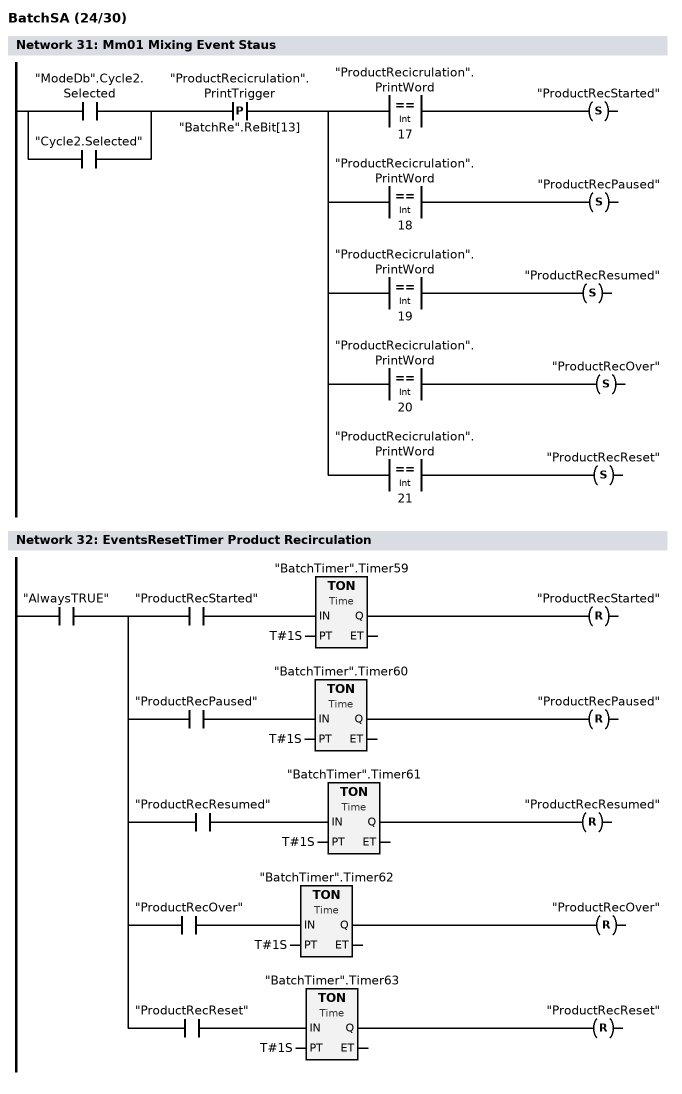
   RUNG wire#powerrail
      Contact( "ModeDb".Cycle2.Selected )
      wire#w1
      P_Contact(operand := "ProductRecicrulation".PrintTrigger, bit := "BatchRe".ReBit[13])
      wire#w2
      { S7_Templates := "SrcType := Int" } EQ_Contact(in1 := "ProductRecicrulation".PrintWord, in2 := 17)
      S_Coil( "ProductRecStarted" )
   END_RUNG
   RUNG wire#powerrail
      Contact( "Cycle2.Selected" )
   END_RUNG wire#w1
   RUNG wire#w2
      { S7_Templates := "SrcType := Int" } EQ_Contact(in1 := "ProductRecicrulation".PrintWord, in2 := 18)
      S_Coil( "ProductRecPaused" )
   END_RUNG
   RUNG wire#w2
      { S7_Templates := "SrcType := Int" } EQ_Contact(in1 := "ProductRecicrulation".PrintWord, in2 := 19)
      S_Coil( "ProductRecResumed" )
   END_RUNG
   RUNG wire#w2
      { S7_Templates := "SrcType := Int" } EQ_Contact(in1 := "ProductRecicrulation".PrintWord, in2 := 20)
      S_Coil( "ProductRecOver" )
   END_RUNG
   RUNG wire#w2
      { S7_Templates := "SrcType := Int" } EQ_Contact(in1 := "ProductRecicrulation".PrintWord, in2 := 21)
      S_Coil( "ProductRecReset" )
   END_RUNG
   // the same network as SCL:
   #_w1 := ("ModeDb".Cycle2.Selected OR "Cycle2.Selected") AND "ProductRecicrulation".PrintTrigger AND NOT "BatchRe".ReBit[13];   // rising edge of "ProductRecicrulation".PrintTrigger
   "BatchRe".ReBit[13] := "ProductRecicrulation".PrintTrigger;
   IF #_w1 AND ("ProductRecicrulation".PrintWord = 17) THEN "ProductRecStarted" := TRUE; END_IF;
   IF #_w1 AND ("ProductRecicrulation".PrintWord = 18) THEN "ProductRecPaused" := TRUE; END_IF;
   IF #_w1 AND ("ProductRecicrulation".PrintWord = 19) THEN "ProductRecResumed" := TRUE; END_IF;
   IF #_w1 AND ("ProductRecicrulation".PrintWord = 20) THEN "ProductRecOver" := TRUE; END_IF;
   IF #_w1 AND ("ProductRecicrulation".PrintWord = 21) THEN "ProductRecReset" := TRUE; END_IF;
END_REGION

REGION Network 32: EventsResetTimer Product Recirculation
   RUNG wire#powerrail
      Contact( "AlwaysTRUE" )
      wire#w1
      Contact( "ProductRecStarted" )
      { S7_Templates := "time_type := Time" } "BatchTimer".Timer59.TON(pt := T#1S, et =>)
      R_Coil( "ProductRecStarted" )
   END_RUNG
   RUNG wire#w1
      Contact( "ProductRecPaused" )
      { S7_Templates := "time_type := Time" } "BatchTimer".Timer60.TON(pt := T#1S, et =>)
      R_Coil( "ProductRecPaused" )
   END_RUNG
   RUNG wire#w1
      Contact( "ProductRecResumed" )
      { S7_Templates := "time_type := Time" } "BatchTimer".Timer61.TON(pt := T#1S, et =>)
      R_Coil( "ProductRecResumed" )
   END_RUNG
   RUNG wire#w1
      Contact( "ProductRecOver" )
      { S7_Templates := "time_type := Time" } "BatchTimer".Timer62.TON(pt := T#1S, et =>)
      R_Coil( "ProductRecOver" )
   END_RUNG
   RUNG wire#w1
      Contact( "ProductRecReset" )
      { S7_Templates := "time_type := Time" } "BatchTimer".Timer63.TON(pt := T#1S, et =>)
      R_Coil( "ProductRecReset" )
   END_RUNG
   // the same network as SCL:
   "BatchTimer".Timer59.TON(IN := "AlwaysTRUE" AND "ProductRecStarted", PT := T#1S);
   IF "BatchTimer".Timer59.Q THEN "ProductRecStarted" := FALSE; END_IF;
   "BatchTimer".Timer60.TON(IN := "AlwaysTRUE" AND "ProductRecPaused", PT := T#1S);
   IF "BatchTimer".Timer60.Q THEN "ProductRecPaused" := FALSE; END_IF;
   "BatchTimer".Timer61.TON(IN := "AlwaysTRUE" AND "ProductRecResumed", PT := T#1S);
   IF "BatchTimer".Timer61.Q THEN "ProductRecResumed" := FALSE; END_IF;
   "BatchTimer".Timer62.TON(IN := "AlwaysTRUE" AND "ProductRecOver", PT := T#1S);
   IF "BatchTimer".Timer62.Q THEN "ProductRecOver" := FALSE; END_IF;
   "BatchTimer".Timer63.TON(IN := "AlwaysTRUE" AND "ProductRecReset", PT := T#1S);
   IF "BatchTimer".Timer63.Q THEN "ProductRecReset" := FALSE; END_IF;
END_REGION

REGION Network 33: EventsResetTimer FIill PWI
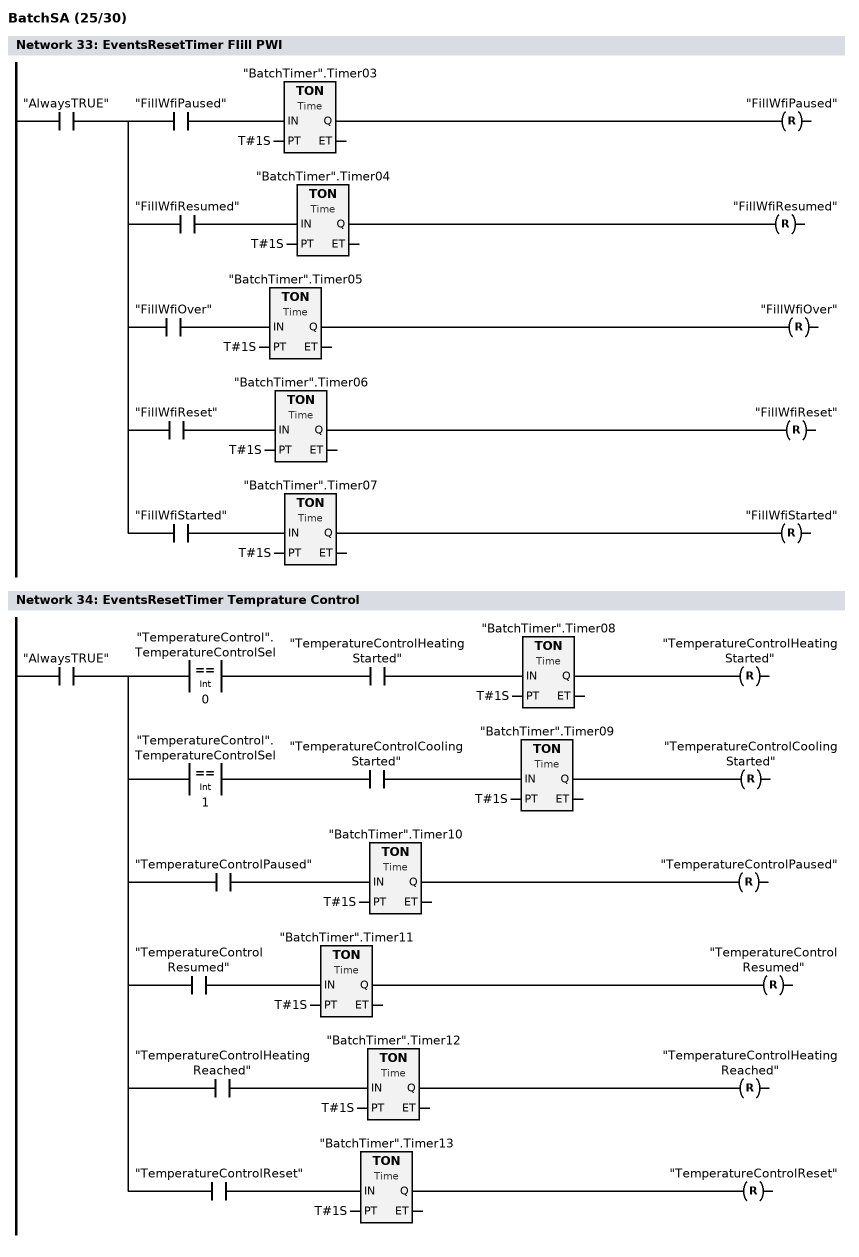
   RUNG wire#powerrail
      Contact( "AlwaysTRUE" )
      wire#w1
      Contact( "FillWfiPaused" )
      { S7_Templates := "time_type := Time" } "BatchTimer".Timer03.TON(pt := T#1S, et =>)
      R_Coil( "FillWfiPaused" )
   END_RUNG
   RUNG wire#w1
      Contact( "FillWfiResumed" )
      { S7_Templates := "time_type := Time" } "BatchTimer".Timer04.TON(pt := T#1S, et =>)
      R_Coil( "FillWfiResumed" )
   END_RUNG
   RUNG wire#w1
      Contact( "FillWfiOver" )
      { S7_Templates := "time_type := Time" } "BatchTimer".Timer05.TON(pt := T#1S, et =>)
      R_Coil( "FillWfiOver" )
   END_RUNG
   RUNG wire#w1
      Contact( "FillWfiReset" )
      { S7_Templates := "time_type := Time" } "BatchTimer".Timer06.TON(pt := T#1S, et =>)
      R_Coil( "FillWfiReset" )
   END_RUNG
   RUNG wire#w1
      Contact( "FillWfiStarted" )
      { S7_Templates := "time_type := Time" } "BatchTimer".Timer07.TON(pt := T#1S, et =>)
      R_Coil( "FillWfiStarted" )
   END_RUNG
   // the same network as SCL:
   "BatchTimer".Timer03.TON(IN := "AlwaysTRUE" AND "FillWfiPaused", PT := T#1S);
   IF "BatchTimer".Timer03.Q THEN "FillWfiPaused" := FALSE; END_IF;
   "BatchTimer".Timer04.TON(IN := "AlwaysTRUE" AND "FillWfiResumed", PT := T#1S);
   IF "BatchTimer".Timer04.Q THEN "FillWfiResumed" := FALSE; END_IF;
   "BatchTimer".Timer05.TON(IN := "AlwaysTRUE" AND "FillWfiOver", PT := T#1S);
   IF "BatchTimer".Timer05.Q THEN "FillWfiOver" := FALSE; END_IF;
   "BatchTimer".Timer06.TON(IN := "AlwaysTRUE" AND "FillWfiReset", PT := T#1S);
   IF "BatchTimer".Timer06.Q THEN "FillWfiReset" := FALSE; END_IF;
   "BatchTimer".Timer07.TON(IN := "AlwaysTRUE" AND "FillWfiStarted", PT := T#1S);
   IF "BatchTimer".Timer07.Q THEN "FillWfiStarted" := FALSE; END_IF;
END_REGION

REGION Network 34: EventsResetTimer Temprature Control
   RUNG wire#powerrail
      Contact( "AlwaysTRUE" )
      wire#w1
      { S7_Templates := "SrcType := Int" } EQ_Contact(in1 := "TemperatureControl".TemperatureControlSel, in2 := 0)
      Contact( "TemperatureControlHeatingStarted" )
      { S7_Templates := "time_type := Time" } "BatchTimer".Timer08.TON(pt := T#1S, et =>)
      R_Coil( "TemperatureControlHeatingStarted" )
   END_RUNG
   RUNG wire#w1
      { S7_Templates := "SrcType := Int" } EQ_Contact(in1 := "TemperatureControl".TemperatureControlSel, in2 := 1)
      Contact( "TemperatureControlCoolingStarted" )
      { S7_Templates := "time_type := Time" } "BatchTimer".Timer09.TON(pt := T#1S, et =>)
      R_Coil( "TemperatureControlCoolingStarted" )
   END_RUNG
   RUNG wire#w1
      Contact( "TemperatureControlPaused" )
      { S7_Templates := "time_type := Time" } "BatchTimer".Timer10.TON(pt := T#1S, et =>)
      R_Coil( "TemperatureControlPaused" )
   END_RUNG
   RUNG wire#w1
      Contact( "TemperatureControlResumed" )
      { S7_Templates := "time_type := Time" } "BatchTimer".Timer11.TON(pt := T#1S, et =>)
      R_Coil( "TemperatureControlResumed" )
   END_RUNG
   RUNG wire#w1
      Contact( "TemperatureControlHeatingReached" )
      { S7_Templates := "time_type := Time" } "BatchTimer".Timer12.TON(pt := T#1S, et =>)
      R_Coil( "TemperatureControlHeatingReached" )
   END_RUNG
   RUNG wire#w1
      Contact( "TemperatureControlReset" )
      { S7_Templates := "time_type := Time" } "BatchTimer".Timer13.TON(pt := T#1S, et =>)
      R_Coil( "TemperatureControlReset" )
   END_RUNG
   // the same network as SCL:
   "BatchTimer".Timer08.TON(IN := "AlwaysTRUE" AND ("TemperatureControl".TemperatureControlSel = 0) AND "TemperatureControlHeatingStarted",
                           PT := T#1S);
   IF "BatchTimer".Timer08.Q THEN "TemperatureControlHeatingStarted" := FALSE; END_IF;
   "BatchTimer".Timer09.TON(IN := "AlwaysTRUE" AND ("TemperatureControl".TemperatureControlSel = 1) AND "TemperatureControlCoolingStarted",
                           PT := T#1S);
   IF "BatchTimer".Timer09.Q THEN "TemperatureControlCoolingStarted" := FALSE; END_IF;
   "BatchTimer".Timer10.TON(IN := "AlwaysTRUE" AND "TemperatureControlPaused", PT := T#1S);
   IF "BatchTimer".Timer10.Q THEN "TemperatureControlPaused" := FALSE; END_IF;
   "BatchTimer".Timer11.TON(IN := "AlwaysTRUE" AND "TemperatureControlResumed", PT := T#1S);
   IF "BatchTimer".Timer11.Q THEN "TemperatureControlResumed" := FALSE; END_IF;
   "BatchTimer".Timer12.TON(IN := "AlwaysTRUE" AND "TemperatureControlHeatingReached", PT := T#1S);
   IF "BatchTimer".Timer12.Q THEN "TemperatureControlHeatingReached" := FALSE; END_IF;
   "BatchTimer".Timer13.TON(IN := "AlwaysTRUE" AND "TemperatureControlReset", PT := T#1S);
   IF "BatchTimer".Timer13.Q THEN "TemperatureControlReset" := FALSE; END_IF;
END_REGION

REGION Network 35: EventsResetTimer RawMaterialAddition
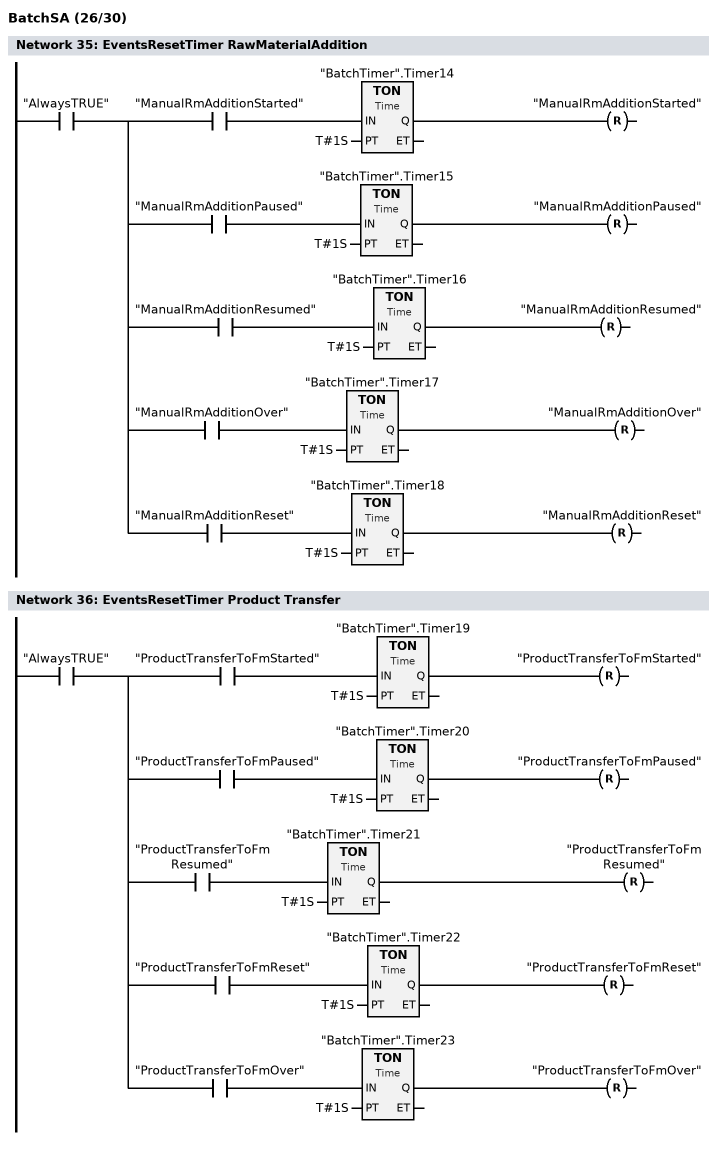
   RUNG wire#powerrail
      Contact( "AlwaysTRUE" )
      wire#w1
      Contact( "ManualRmAdditionStarted" )
      { S7_Templates := "time_type := Time" } "BatchTimer".Timer14.TON(pt := T#1S, et =>)
      R_Coil( "ManualRmAdditionStarted" )
   END_RUNG
   RUNG wire#w1
      Contact( "ManualRmAdditionPaused" )
      { S7_Templates := "time_type := Time" } "BatchTimer".Timer15.TON(pt := T#1S, et =>)
      R_Coil( "ManualRmAdditionPaused" )
   END_RUNG
   RUNG wire#w1
      Contact( "ManualRmAdditionResumed" )
      { S7_Templates := "time_type := Time" } "BatchTimer".Timer16.TON(pt := T#1S, et =>)
      R_Coil( "ManualRmAdditionResumed" )
   END_RUNG
   RUNG wire#w1
      Contact( "ManualRmAdditionOver" )
      { S7_Templates := "time_type := Time" } "BatchTimer".Timer17.TON(pt := T#1S, et =>)
      R_Coil( "ManualRmAdditionOver" )
   END_RUNG
   RUNG wire#w1
      Contact( "ManualRmAdditionReset" )
      { S7_Templates := "time_type := Time" } "BatchTimer".Timer18.TON(pt := T#1S, et =>)
      R_Coil( "ManualRmAdditionReset" )
   END_RUNG
   // the same network as SCL:
   "BatchTimer".Timer14.TON(IN := "AlwaysTRUE" AND "ManualRmAdditionStarted", PT := T#1S);
   IF "BatchTimer".Timer14.Q THEN "ManualRmAdditionStarted" := FALSE; END_IF;
   "BatchTimer".Timer15.TON(IN := "AlwaysTRUE" AND "ManualRmAdditionPaused", PT := T#1S);
   IF "BatchTimer".Timer15.Q THEN "ManualRmAdditionPaused" := FALSE; END_IF;
   "BatchTimer".Timer16.TON(IN := "AlwaysTRUE" AND "ManualRmAdditionResumed", PT := T#1S);
   IF "BatchTimer".Timer16.Q THEN "ManualRmAdditionResumed" := FALSE; END_IF;
   "BatchTimer".Timer17.TON(IN := "AlwaysTRUE" AND "ManualRmAdditionOver", PT := T#1S);
   IF "BatchTimer".Timer17.Q THEN "ManualRmAdditionOver" := FALSE; END_IF;
   "BatchTimer".Timer18.TON(IN := "AlwaysTRUE" AND "ManualRmAdditionReset", PT := T#1S);
   IF "BatchTimer".Timer18.Q THEN "ManualRmAdditionReset" := FALSE; END_IF;
END_REGION

REGION Network 36: EventsResetTimer Product Transfer
   RUNG wire#powerrail
      Contact( "AlwaysTRUE" )
      wire#w1
      Contact( "ProductTransferToFmStarted" )
      { S7_Templates := "time_type := Time" } "BatchTimer".Timer19.TON(pt := T#1S, et =>)
      R_Coil( "ProductTransferToFmStarted" )
   END_RUNG
   RUNG wire#w1
      Contact( "ProductTransferToFmPaused" )
      { S7_Templates := "time_type := Time" } "BatchTimer".Timer20.TON(pt := T#1S, et =>)
      R_Coil( "ProductTransferToFmPaused" )
   END_RUNG
   RUNG wire#w1
      Contact( "ProductTransferToFmResumed" )
      { S7_Templates := "time_type := Time" } "BatchTimer".Timer21.TON(pt := T#1S, et =>)
      R_Coil( "ProductTransferToFmResumed" )
   END_RUNG
   RUNG wire#w1
      Contact( "ProductTransferToFmReset" )
      { S7_Templates := "time_type := Time" } "BatchTimer".Timer22.TON(pt := T#1S, et =>)
      R_Coil( "ProductTransferToFmReset" )
   END_RUNG
   RUNG wire#w1
      Contact( "ProductTransferToFmOver" )
      { S7_Templates := "time_type := Time" } "BatchTimer".Timer23.TON(pt := T#1S, et =>)
      R_Coil( "ProductTransferToFmOver" )
   END_RUNG
   // the same network as SCL:
   "BatchTimer".Timer19.TON(IN := "AlwaysTRUE" AND "ProductTransferToFmStarted", PT := T#1S);
   IF "BatchTimer".Timer19.Q THEN "ProductTransferToFmStarted" := FALSE; END_IF;
   "BatchTimer".Timer20.TON(IN := "AlwaysTRUE" AND "ProductTransferToFmPaused", PT := T#1S);
   IF "BatchTimer".Timer20.Q THEN "ProductTransferToFmPaused" := FALSE; END_IF;
   "BatchTimer".Timer21.TON(IN := "AlwaysTRUE" AND "ProductTransferToFmResumed", PT := T#1S);
   IF "BatchTimer".Timer21.Q THEN "ProductTransferToFmResumed" := FALSE; END_IF;
   "BatchTimer".Timer22.TON(IN := "AlwaysTRUE" AND "ProductTransferToFmReset", PT := T#1S);
   IF "BatchTimer".Timer22.Q THEN "ProductTransferToFmReset" := FALSE; END_IF;
   "BatchTimer".Timer23.TON(IN := "AlwaysTRUE" AND "ProductTransferToFmOver", PT := T#1S);
   IF "BatchTimer".Timer23.Q THEN "ProductTransferToFmOver" := FALSE; END_IF;
END_REGION

REGION Network 37: EventsResetTimer Mm01 Mixing
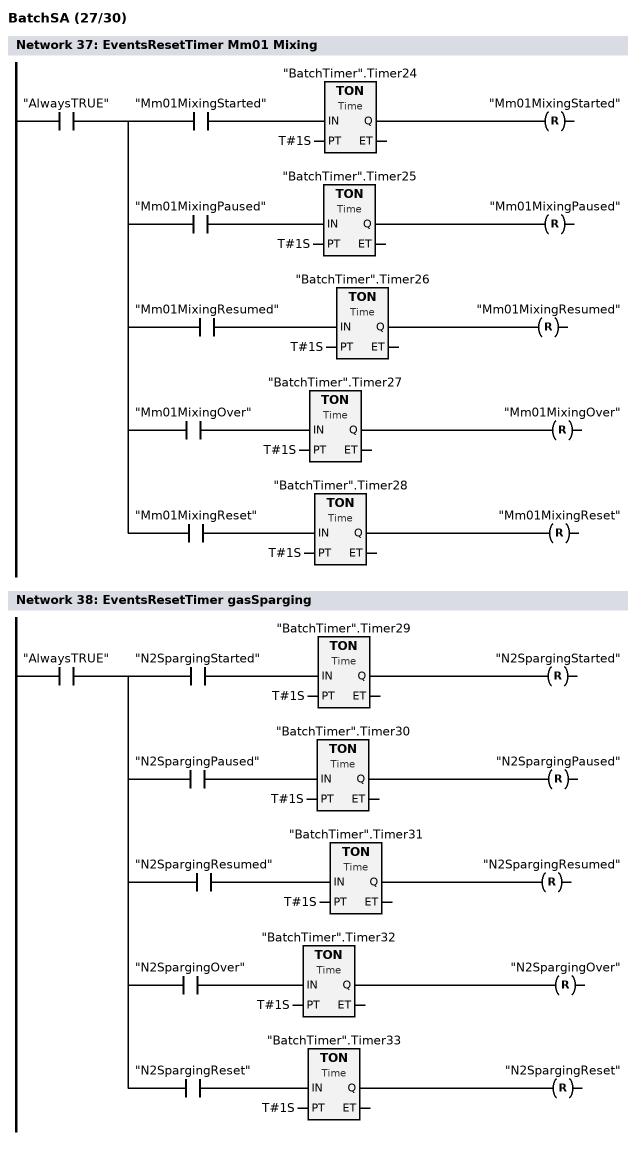
   RUNG wire#powerrail
      Contact( "AlwaysTRUE" )
      wire#w1
      Contact( "Mm01MixingStarted" )
      { S7_Templates := "time_type := Time" } "BatchTimer".Timer24.TON(pt := T#1S, et =>)
      R_Coil( "Mm01MixingStarted" )
   END_RUNG
   RUNG wire#w1
      Contact( "Mm01MixingPaused" )
      { S7_Templates := "time_type := Time" } "BatchTimer".Timer25.TON(pt := T#1S, et =>)
      R_Coil( "Mm01MixingPaused" )
   END_RUNG
   RUNG wire#w1
      Contact( "Mm01MixingResumed" )
      { S7_Templates := "time_type := Time" } "BatchTimer".Timer26.TON(pt := T#1S, et =>)
      R_Coil( "Mm01MixingResumed" )
   END_RUNG
   RUNG wire#w1
      Contact( "Mm01MixingOver" )
      { S7_Templates := "time_type := Time" } "BatchTimer".Timer27.TON(pt := T#1S, et =>)
      R_Coil( "Mm01MixingOver" )
   END_RUNG
   RUNG wire#w1
      Contact( "Mm01MixingReset" )
      { S7_Templates := "time_type := Time" } "BatchTimer".Timer28.TON(pt := T#1S, et =>)
      R_Coil( "Mm01MixingReset" )
   END_RUNG
   // the same network as SCL:
   "BatchTimer".Timer24.TON(IN := "AlwaysTRUE" AND "Mm01MixingStarted", PT := T#1S);
   IF "BatchTimer".Timer24.Q THEN "Mm01MixingStarted" := FALSE; END_IF;
   "BatchTimer".Timer25.TON(IN := "AlwaysTRUE" AND "Mm01MixingPaused", PT := T#1S);
   IF "BatchTimer".Timer25.Q THEN "Mm01MixingPaused" := FALSE; END_IF;
   "BatchTimer".Timer26.TON(IN := "AlwaysTRUE" AND "Mm01MixingResumed", PT := T#1S);
   IF "BatchTimer".Timer26.Q THEN "Mm01MixingResumed" := FALSE; END_IF;
   "BatchTimer".Timer27.TON(IN := "AlwaysTRUE" AND "Mm01MixingOver", PT := T#1S);
   IF "BatchTimer".Timer27.Q THEN "Mm01MixingOver" := FALSE; END_IF;
   "BatchTimer".Timer28.TON(IN := "AlwaysTRUE" AND "Mm01MixingReset", PT := T#1S);
   IF "BatchTimer".Timer28.Q THEN "Mm01MixingReset" := FALSE; END_IF;
END_REGION

REGION Network 38: EventsResetTimer gasSparging
   RUNG wire#powerrail
      Contact( "AlwaysTRUE" )
      wire#w1
      Contact( "N2SpargingStarted" )
      { S7_Templates := "time_type := Time" } "BatchTimer".Timer29.TON(pt := T#1S, et =>)
      R_Coil( "N2SpargingStarted" )
   END_RUNG
   RUNG wire#w1
      Contact( "N2SpargingPaused" )
      { S7_Templates := "time_type := Time" } "BatchTimer".Timer30.TON(pt := T#1S, et =>)
      R_Coil( "N2SpargingPaused" )
   END_RUNG
   RUNG wire#w1
      Contact( "N2SpargingResumed" )
      { S7_Templates := "time_type := Time" } "BatchTimer".Timer31.TON(pt := T#1S, et =>)
      R_Coil( "N2SpargingResumed" )
   END_RUNG
   RUNG wire#w1
      Contact( "N2SpargingOver" )
      { S7_Templates := "time_type := Time" } "BatchTimer".Timer32.TON(pt := T#1S, et =>)
      R_Coil( "N2SpargingOver" )
   END_RUNG
   RUNG wire#w1
      Contact( "N2SpargingReset" )
      { S7_Templates := "time_type := Time" } "BatchTimer".Timer33.TON(pt := T#1S, et =>)
      R_Coil( "N2SpargingReset" )
   END_RUNG
   // the same network as SCL:
   "BatchTimer".Timer29.TON(IN := "AlwaysTRUE" AND "N2SpargingStarted", PT := T#1S);
   IF "BatchTimer".Timer29.Q THEN "N2SpargingStarted" := FALSE; END_IF;
   "BatchTimer".Timer30.TON(IN := "AlwaysTRUE" AND "N2SpargingPaused", PT := T#1S);
   IF "BatchTimer".Timer30.Q THEN "N2SpargingPaused" := FALSE; END_IF;
   "BatchTimer".Timer31.TON(IN := "AlwaysTRUE" AND "N2SpargingResumed", PT := T#1S);
   IF "BatchTimer".Timer31.Q THEN "N2SpargingResumed" := FALSE; END_IF;
   "BatchTimer".Timer32.TON(IN := "AlwaysTRUE" AND "N2SpargingOver", PT := T#1S);
   IF "BatchTimer".Timer32.Q THEN "N2SpargingOver" := FALSE; END_IF;
   "BatchTimer".Timer33.TON(IN := "AlwaysTRUE" AND "N2SpargingReset", PT := T#1S);
   IF "BatchTimer".Timer33.Q THEN "N2SpargingReset" := FALSE; END_IF;
END_REGION

REGION Network 39: EventsResetTimer Gas Blanketing
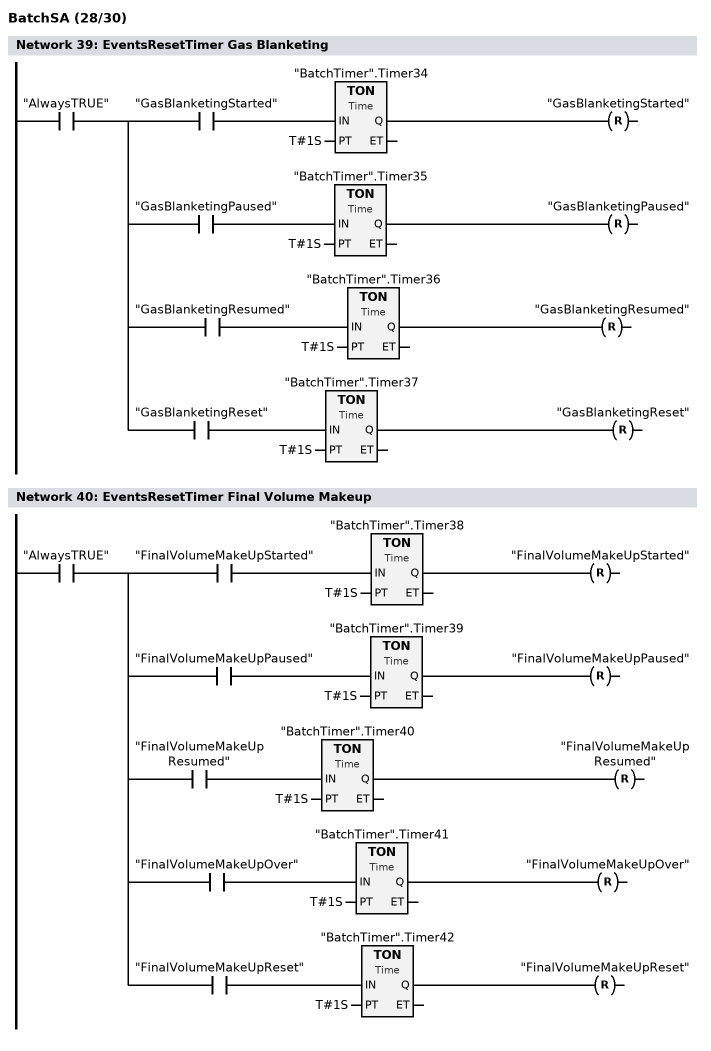
   RUNG wire#powerrail
      Contact( "AlwaysTRUE" )
      wire#w1
      Contact( "GasBlanketingStarted" )
      { S7_Templates := "time_type := Time" } "BatchTimer".Timer34.TON(pt := T#1S, et =>)
      R_Coil( "GasBlanketingStarted" )
   END_RUNG
   RUNG wire#w1
      Contact( "GasBlanketingPaused" )
      { S7_Templates := "time_type := Time" } "BatchTimer".Timer35.TON(pt := T#1S, et =>)
      R_Coil( "GasBlanketingPaused" )
   END_RUNG
   RUNG wire#w1
      Contact( "GasBlanketingResumed" )
      { S7_Templates := "time_type := Time" } "BatchTimer".Timer36.TON(pt := T#1S, et =>)
      R_Coil( "GasBlanketingResumed" )
   END_RUNG
   RUNG wire#w1
      Contact( "GasBlanketingReset" )
      { S7_Templates := "time_type := Time" } "BatchTimer".Timer37.TON(pt := T#1S, et =>)
      R_Coil( "GasBlanketingReset" )
   END_RUNG
   // the same network as SCL:
   "BatchTimer".Timer34.TON(IN := "AlwaysTRUE" AND "GasBlanketingStarted", PT := T#1S);
   IF "BatchTimer".Timer34.Q THEN "GasBlanketingStarted" := FALSE; END_IF;
   "BatchTimer".Timer35.TON(IN := "AlwaysTRUE" AND "GasBlanketingPaused", PT := T#1S);
   IF "BatchTimer".Timer35.Q THEN "GasBlanketingPaused" := FALSE; END_IF;
   "BatchTimer".Timer36.TON(IN := "AlwaysTRUE" AND "GasBlanketingResumed", PT := T#1S);
   IF "BatchTimer".Timer36.Q THEN "GasBlanketingResumed" := FALSE; END_IF;
   "BatchTimer".Timer37.TON(IN := "AlwaysTRUE" AND "GasBlanketingReset", PT := T#1S);
   IF "BatchTimer".Timer37.Q THEN "GasBlanketingReset" := FALSE; END_IF;
END_REGION

REGION Network 40: EventsResetTimer Final Volume Makeup
   RUNG wire#powerrail
      Contact( "AlwaysTRUE" )
      wire#w1
      Contact( "FinalVolumeMakeUpStarted" )
      { S7_Templates := "time_type := Time" } "BatchTimer".Timer38.TON(pt := T#1S, et =>)
      R_Coil( "FinalVolumeMakeUpStarted" )
   END_RUNG
   RUNG wire#w1
      Contact( "FinalVolumeMakeUpPaused" )
      { S7_Templates := "time_type := Time" } "BatchTimer".Timer39.TON(pt := T#1S, et =>)
      R_Coil( "FinalVolumeMakeUpPaused" )
   END_RUNG
   RUNG wire#w1
      Contact( "FinalVolumeMakeUpResumed" )
      { S7_Templates := "time_type := Time" } "BatchTimer".Timer40.TON(pt := T#1S, et =>)
      R_Coil( "FinalVolumeMakeUpResumed" )
   END_RUNG
   RUNG wire#w1
      Contact( "FinalVolumeMakeUpOver" )
      { S7_Templates := "time_type := Time" } "BatchTimer".Timer41.TON(pt := T#1S, et =>)
      R_Coil( "FinalVolumeMakeUpOver" )
   END_RUNG
   RUNG wire#w1
      Contact( "FinalVolumeMakeUpReset" )
      { S7_Templates := "time_type := Time" } "BatchTimer".Timer42.TON(pt := T#1S, et =>)
      R_Coil( "FinalVolumeMakeUpReset" )
   END_RUNG
   // the same network as SCL:
   "BatchTimer".Timer38.TON(IN := "AlwaysTRUE" AND "FinalVolumeMakeUpStarted", PT := T#1S);
   IF "BatchTimer".Timer38.Q THEN "FinalVolumeMakeUpStarted" := FALSE; END_IF;
   "BatchTimer".Timer39.TON(IN := "AlwaysTRUE" AND "FinalVolumeMakeUpPaused", PT := T#1S);
   IF "BatchTimer".Timer39.Q THEN "FinalVolumeMakeUpPaused" := FALSE; END_IF;
   "BatchTimer".Timer40.TON(IN := "AlwaysTRUE" AND "FinalVolumeMakeUpResumed", PT := T#1S);
   IF "BatchTimer".Timer40.Q THEN "FinalVolumeMakeUpResumed" := FALSE; END_IF;
   "BatchTimer".Timer41.TON(IN := "AlwaysTRUE" AND "FinalVolumeMakeUpOver", PT := T#1S);
   IF "BatchTimer".Timer41.Q THEN "FinalVolumeMakeUpOver" := FALSE; END_IF;
   "BatchTimer".Timer42.TON(IN := "AlwaysTRUE" AND "FinalVolumeMakeUpReset", PT := T#1S);
   IF "BatchTimer".Timer42.Q THEN "FinalVolumeMakeUpReset" := FALSE; END_IF;
END_REGION

REGION Network 41: EventsResetTimer Jacket
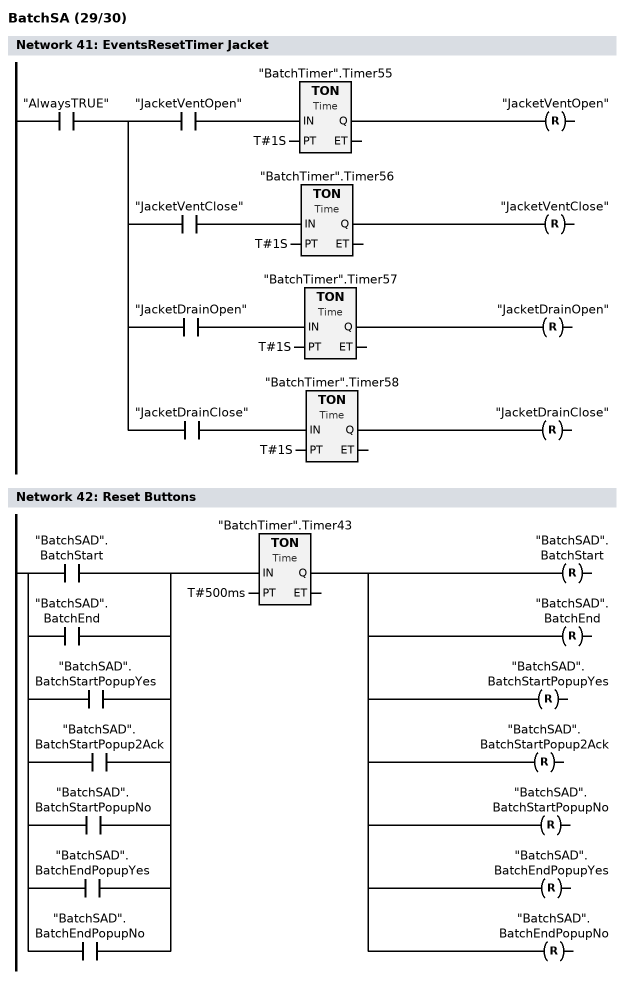
   RUNG wire#powerrail
      Contact( "AlwaysTRUE" )
      wire#w1
      Contact( "JacketVentOpen" )
      { S7_Templates := "time_type := Time" } "BatchTimer".Timer55.TON(pt := T#1S, et =>)
      R_Coil( "JacketVentOpen" )
   END_RUNG
   RUNG wire#w1
      Contact( "JacketVentClose" )
      { S7_Templates := "time_type := Time" } "BatchTimer".Timer56.TON(pt := T#1S, et =>)
      R_Coil( "JacketVentClose" )
   END_RUNG
   RUNG wire#w1
      Contact( "JacketDrainOpen" )
      { S7_Templates := "time_type := Time" } "BatchTimer".Timer57.TON(pt := T#1S, et =>)
      R_Coil( "JacketDrainOpen" )
   END_RUNG
   RUNG wire#w1
      Contact( "JacketDrainClose" )
      { S7_Templates := "time_type := Time" } "BatchTimer".Timer58.TON(pt := T#1S, et =>)
      R_Coil( "JacketDrainClose" )
   END_RUNG
   // the same network as SCL:
   "BatchTimer".Timer55.TON(IN := "AlwaysTRUE" AND "JacketVentOpen", PT := T#1S);
   IF "BatchTimer".Timer55.Q THEN "JacketVentOpen" := FALSE; END_IF;
   "BatchTimer".Timer56.TON(IN := "AlwaysTRUE" AND "JacketVentClose", PT := T#1S);
   IF "BatchTimer".Timer56.Q THEN "JacketVentClose" := FALSE; END_IF;
   "BatchTimer".Timer57.TON(IN := "AlwaysTRUE" AND "JacketDrainOpen", PT := T#1S);
   IF "BatchTimer".Timer57.Q THEN "JacketDrainOpen" := FALSE; END_IF;
   "BatchTimer".Timer58.TON(IN := "AlwaysTRUE" AND "JacketDrainClose", PT := T#1S);
   IF "BatchTimer".Timer58.Q THEN "JacketDrainClose" := FALSE; END_IF;
END_REGION

REGION Network 42: Reset Buttons
   RUNG wire#powerrail
      Contact( "BatchSAD".BatchStart )
      wire#w1
      { S7_Templates := "time_type := Time" } "BatchTimer".Timer43.TON(pt := T#500ms, et =>)
      wire#w2
      R_Coil( "BatchSAD".BatchStart )
   END_RUNG
   RUNG wire#powerrail
      Contact( "BatchSAD".BatchEnd )
   END_RUNG wire#w1
   RUNG wire#powerrail
      Contact( "BatchSAD".BatchStartPopupYes )
   END_RUNG wire#w1
   RUNG wire#powerrail
      Contact( "BatchSAD".BatchStartPopup2Ack )
   END_RUNG wire#w1
   RUNG wire#powerrail
      Contact( "BatchSAD".BatchStartPopupNo )
   END_RUNG wire#w1
   RUNG wire#powerrail
      Contact( "BatchSAD".BatchEndPopupYes )
   END_RUNG wire#w1
   RUNG wire#powerrail
      Contact( "BatchSAD".BatchEndPopupNo )
   END_RUNG wire#w1
   RUNG wire#w2
      R_Coil( "BatchSAD".BatchEnd )
   END_RUNG
   RUNG wire#w2
      R_Coil( "BatchSAD".BatchStartPopupYes )
   END_RUNG
   RUNG wire#w2
      R_Coil( "BatchSAD".BatchStartPopup2Ack )
   END_RUNG
   RUNG wire#w2
      R_Coil( "BatchSAD".BatchStartPopupNo )
   END_RUNG
   RUNG wire#w2
      R_Coil( "BatchSAD".BatchEndPopupYes )
   END_RUNG
   RUNG wire#w2
      R_Coil( "BatchSAD".BatchEndPopupNo )
   END_RUNG
   // the same network as SCL:
   "BatchTimer".Timer43.TON(IN := "BatchSAD".BatchStart OR "BatchSAD".BatchEnd OR "BatchSAD".BatchStartPopupYes OR "BatchSAD".BatchStartPopup2Ack OR "BatchSAD".BatchStartPopupNo OR "BatchSAD".BatchEndPopupYes OR "BatchSAD".BatchEndPopupNo,
                           PT := T#500ms);
   IF "BatchTimer".Timer43.Q THEN
       "BatchSAD".BatchStart := FALSE;
       "BatchSAD".BatchEnd := FALSE;
       "BatchSAD".BatchStartPopupYes := FALSE;
       "BatchSAD".BatchStartPopup2Ack := FALSE;
       "BatchSAD".BatchStartPopupNo := FALSE;
       "BatchSAD".BatchEndPopupYes := FALSE;
       "BatchSAD".BatchEndPopupNo := FALSE;
   END_IF;
END_REGION

REGION Network 43: RESET
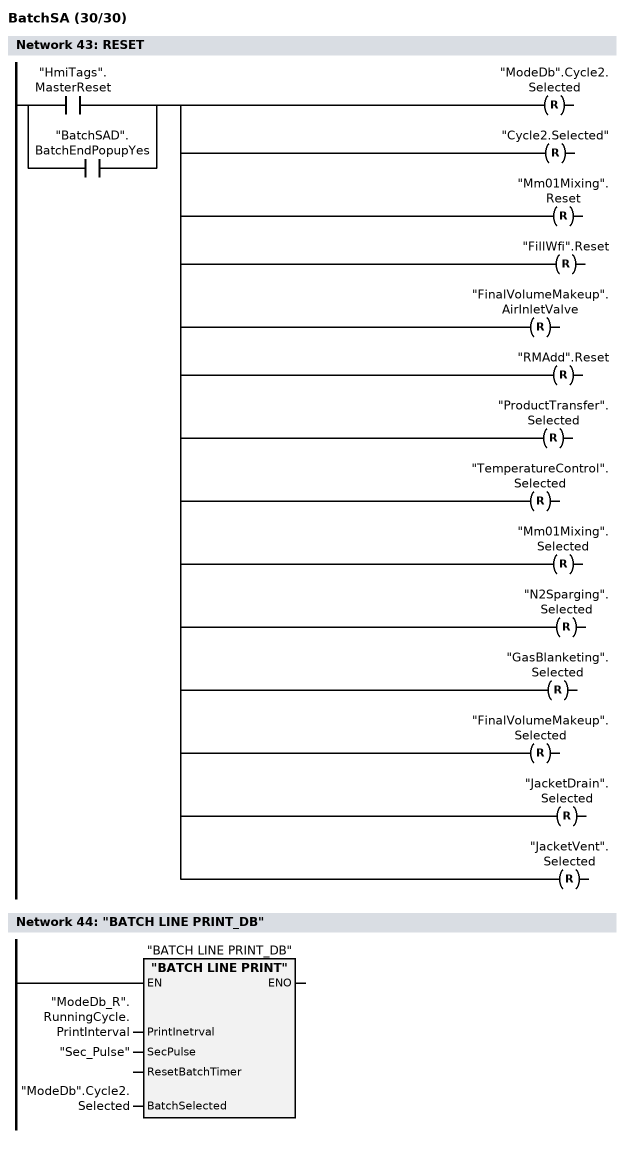
   RUNG wire#powerrail
      Contact( "HmiTags".MasterReset )
      wire#w1
      R_Coil( "ModeDb".Cycle2.Selected )
   END_RUNG
   RUNG wire#powerrail
      Contact( "BatchSAD".BatchEndPopupYes )
   END_RUNG wire#w1
   RUNG wire#w1
      R_Coil( "Cycle2.Selected" )
   END_RUNG
   RUNG wire#w1
      R_Coil( "Mm01Mixing".Reset )
   END_RUNG
   RUNG wire#w1
      R_Coil( "FillWfi".Reset )
   END_RUNG
   RUNG wire#w1
      R_Coil( "FinalVolumeMakeup".AirInletValve )
   END_RUNG
   RUNG wire#w1
      R_Coil( "RMAdd".Reset )
   END_RUNG
   RUNG wire#w1
      R_Coil( "ProductTransfer".Selected )
   END_RUNG
   RUNG wire#w1
      R_Coil( "TemperatureControl".Selected )
   END_RUNG
   RUNG wire#w1
      R_Coil( "Mm01Mixing".Selected )
   END_RUNG
   RUNG wire#w1
      R_Coil( "N2Sparging".Selected )
   END_RUNG
   RUNG wire#w1
      R_Coil( "GasBlanketing".Selected )
   END_RUNG
   RUNG wire#w1
      R_Coil( "FinalVolumeMakeup".Selected )
   END_RUNG
   RUNG wire#w1
      R_Coil( "JacketDrain".Selected )
   END_RUNG
   RUNG wire#w1
      R_Coil( "JacketVent".Selected )
   END_RUNG
   // the same network as SCL:
   IF "HmiTags".MasterReset OR "BatchSAD".BatchEndPopupYes THEN
       "ModeDb".Cycle2.Selected := FALSE;
       "Cycle2.Selected" := FALSE;
       "Mm01Mixing".Reset := FALSE;
       "FillWfi".Reset := FALSE;
       "FinalVolumeMakeup".AirInletValve := FALSE;
       "RMAdd".Reset := FALSE;
       "ProductTransfer".Selected := FALSE;
       "TemperatureControl".Selected := FALSE;
       "Mm01Mixing".Selected := FALSE;
       "N2Sparging".Selected := FALSE;
       "GasBlanketing".Selected := FALSE;
       "FinalVolumeMakeup".Selected := FALSE;
       "JacketDrain".Selected := FALSE;
       "JacketVent".Selected := FALSE;
   END_IF;
END_REGION

REGION Network 44: "BATCH LINE PRINT_DB"
   RUNG wire#powerrail
      "BATCH LINE PRINT_DB"(PrintInetrval := "ModeDb_R".RunningCycle.PrintInterval, SecPulse := "Sec_Pulse", ResetBatchTimer :=, BatchSelected := "ModeDb".Cycle2.Selected)
   END_RUNG
   // the same network as SCL:
   "BATCH LINE PRINT_DB"(PrintInetrval := "ModeDb_R".RunningCycle.PrintInterval,   // "BATCH LINE PRINT"
                         SecPulse := "Sec_Pulse",
                         BatchSelected := "ModeDb".Cycle2.Selected);
END_REGION
END_FUNCTION
